{attribute addProperty BoxType "EK1100-0000-0018"}
{attribute addProperty Id "Beckhoff_ELM3xxxEK1122Beckhoff_ELM3xxxEK1122_52A3E13B162A_0001_ELM3002_0000_0016ELM3002_08F8D9E433842.25A_0002_ELM3002_0000_0017ELM3002_08F8D9E433842.25A_0003_ELM3002_0000_0018ELM3002_08F8D9E433842.25A_0004_ELM3004_0000_0016ELM3004_B740F21646658.25A_0005_ELM3004_0000_0017ELM3004_B740F21646658.25A_0006_ELM3004_0000_0018ELM3004_B740F21646658.25A_0007_ELM3004_0000_0019ELM3004_B740F21646658.25"}
{attribute addProperty CRC "1858388275"}
{attribute addProperty SizeInBites "2894"}
{attribute addProperty SizeInBytes "361.75"}
TYPE Beckhoff_ELM3xxx_6EC4C133 EXTENDS EK1100_179A0949 :
STRUCT
	{attribute addProperty Name "Beckhoff_ELM3xxxEK1122"}
	Beckhoff_ELM3xxxEK1122 : Beckhoff_ELM3xxxEK1122_52A3E13B;
	{attribute addProperty Name "A_0001_ELM3002_0000_0016"}
	A_0001_ELM3002_0000_0016 : ELM3002_08F8D9E4;
	{attribute addProperty Name "A_0002_ELM3002_0000_0017"}
	A_0002_ELM3002_0000_0017 : ELM3002_08F8D9E4;
	{attribute addProperty Name "A_0003_ELM3002_0000_0018"}
	A_0003_ELM3002_0000_0018 : ELM3002_08F8D9E4;
	{attribute addProperty Name "A_0004_ELM3004_0000_0016"}
	A_0004_ELM3004_0000_0016 : ELM3004_B740F216;
	{attribute addProperty Name "A_0005_ELM3004_0000_0017"}
	A_0005_ELM3004_0000_0017 : ELM3004_B740F216;
	{attribute addProperty Name "A_0006_ELM3004_0000_0018"}
	A_0006_ELM3004_0000_0018 : ELM3004_B740F216;
	{attribute addProperty Name "A_0007_ELM3004_0000_0019"}
	A_0007_ELM3004_0000_0019 : ELM3004_B740F216;
END_STRUCT
END_TYPE

(* stored: Version 1.2.0.0, ProductVersion 3.1.4024.9
   DUT Beckhoff_ELM3xxx_6EC4C133: Id {445e2289-79be-4182-9401-02e5b39bdbde} *)
